TYPE ST_CylinderX_Command :
    STRUCT
        RetractExtend  : BOOL;
        RetractCylinder : BOOL;
    END_STRUCT
END_TYPE

(* stored: Version 1.1.0.1
   DUT ST_CylinderX_Command: Id {d44409e6-319f-4e95-a8f4-c35c15ab4350} *)
